FUNCTION_BLOCK CurrentFloor (* Basic Function Block Type *)
  (* Standard: 61499-2 *)
  (* Version 0.0, 9/23/2026, macie, Schneider Electric, Template *)
  PACKAGE Main;
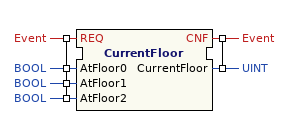
  EVENT_INPUT
    REQ WITH AtFloor0, AtFloor1, AtFloor2; (* Normal Execution Request *)
  END_EVENT
  EVENT_OUTPUT
    CNF WITH CurrentFloor; (* Execution Confirmation *)
  END_EVENT
  VAR_INPUT
    AtFloor0 : BOOL; (* Input event qualifier *)
    AtFloor1 : BOOL;
    AtFloor2 : BOOL;
  END_VAR
  VAR_OUTPUT
    CurrentFloor : UINT := 2; (* Output event qualifier *)
  END_VAR
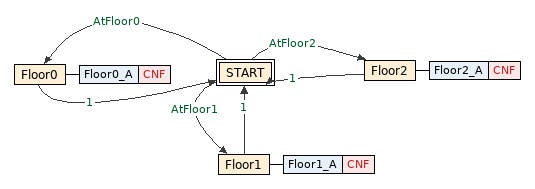
  EC_STATES
    START; (* Initial State *)
    Floor0 : Floor0_A -> CNF;
    Floor1 : Floor1_A -> CNF;
    Floor2 : Floor2_A -> CNF;
  END_STATES
  EC_TRANSITIONS
    START TO Floor2 := AtFloor2;
    Floor2 TO START := 1;
    START TO Floor1 := AtFloor1;
    Floor1 TO START := 1;
    START TO Floor0 := AtFloor0;
    Floor0 TO START := 1;
  END_TRANSITIONS
  ALGORITHM Floor0_A IN ST: (* Initialization algorithm *)
;
CurrentFloor := 0;
  END_ALGORITHM
  ALGORITHM Floor1_A IN ST: (* Normally executed algorithm *)
;
CurrentFloor := 1;
  END_ALGORITHM
  ALGORITHM Floor2_A IN ST:
CurrentFloor := 2;
  END_ALGORITHM
END_FUNCTION_BLOCK
